Fanuc KAREL source: ks00031.KL

-- PROVISIONAL review KL for V940-1; original PC SHA256 9f35586b00e4672845e92c3abc4adddae5297edf78e6719c5708d39e397894ab
-- Incomplete behavior may be omitted. Consult companion uncertainty JSON. Do not deploy.
PROGRAM KS00031
%NOLOCKGROUP
VAR
  FLAG : BOOLEAN
  N : INTEGER
  STATUS : INTEGER
  PN : STRING[80]
  VN : STRING[80]
-- UNRESOLVED_DECL A type=00201c
-- UNRESOLVED_DECL B type=00201c
BEGIN
  -- V9_ZERO_TABLE_METADATA_HINT layout=0001; no indexed target words; source/name/runtime held
  -- UNRESOLVED_PC offsets 5-13; opcodes 3F,75
  -- UNRESOLVED_PC offsets 18-27; opcodes 3F,75
  -- UNRESOLVED_PC offsets 32-46; opcodes 22,22,1E
  -- UNRESOLVED_PC offsets 51-55; opcodes 7F
END KS00031
